// TIA Portal V20 export
VAR_GLOBAL   // PLC tag table "08_CmInfo"
END_VAR
VAR_GLOBAL CONSTANT   // user constants
   NO_OF_RF_IDENT_DEVICES : USInt := 0;   // SICAR: Anzahl der RF Lesestellen / SICAR: Number of RF readers
   NO_OF_RF_ANTENNA_DEVICES : USInt := 2;   // SICAR: Number of RF antennas
END_VAR
